PROGRAM MAIN
VAR
	bExecute : BOOL;
	fbEcInitialiseNewSlaveCountTopology : FB_EcInitialiseNewSlaveCountTopology;
END_VAR

fbEcInitialiseNewSlaveCountTopology(
	stMasterNetIdPhys:=stMasterNetIdPhys, 
	bEnable:= TRUE, 
	bExecute:= bExecute , 
	tTimeout:= , 
	bBusy=> , 
	bError=> , 
	nErrId=> );

bExecute := FALSE;

END_PROGRAM

(* stored: Version 1.1.0.1, ProductVersion 3.1.4024.3
   POU MAIN: Id {b31057fa-aa28-4d9d-bc16-e5b53e7f8556}, SpecialFunc None *)
